{attribute 'qualified_only'}
VAR_GLOBAL
	batch_job_container_creator : FB_BatchJobContainerCreator;
	parallel_job_container_creator : FB_ParallelJobContainerCreator;
	queue_job_container_creator : FB_QueueJobContainerCreator;
	parallel_queue_job_container_creator : FB_ParallelQueueJobContainerCreator;
	axis1	: AXIS_REF;
	axis2	: AXIS_REF;
	motion_command : MotionCommand;
END_VAR

(* stored: Version 1.1.0.1, ProductVersion 3.1.4026.17
   GVL GVL: Id {28486044-a7c6-49b3-93e4-15a4115f2942} *)
